Yaskawa INFORM job: sDrill44_(11).JBI

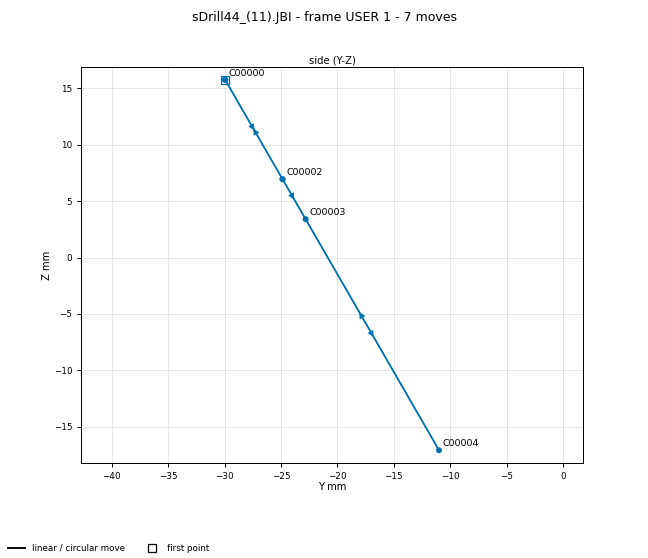
[picture p0: tool path of sDrill44_(11).JBI in frame USER 1, 7 of 7 moves have a stored position in this frame; points joined in program order, loops and branches not executed]
/JOB
//NAME sDrill44_(11)
//POS
///NPOS 7,0,0,0,0,0
///USER 1
///TOOL 3
///POSTYPE USER
///RECTAN
///RCONF 1,0,0,0,0,0
C00000=1.964,-29.946,15.742,-90.000,-150.794,-116.565
C00001=1.964,-29.946,15.742,-90.000,-150.794,-116.565
C00002=1.964,-24.866,6.943,-90.000,-150.794,-116.565
C00003=1.964,-22.817,3.394,-90.000,-150.794,-116.565
C00004=1.964,-11.000,-17.074,-90.000,-150.794,-116.565
C00005=1.964,-24.866,6.943,-90.000,-150.794,-116.565
C00006=1.964,-29.946,15.742,-90.000,-150.794,-116.565
//INST
///ATTR SC,RW,RJ
////FRAME USER 1
///GROUP1 RB1
///LVARS 2,0,0,0,0,0,0,0
NOP
SET LB000 1
SET LB001 25
MOVJ C00000 VJ=17
' Cutting Move Starts
MOVL C00001 V=17 PL=LB000 ACC=LB001 DEC=LB001
MOVL C00002 V=17 PL=LB000 ACC=LB001 DEC=LB001
MOVL C00003 V=17 PL=LB000 ACC=LB001 DEC=LB001
MOVL C00004 V=7 PL=LB000 ACC=LB001 DEC=LB001
MOVL C00005 V=17 PL=LB000 ACC=LB001 DEC=LB001
' Rapid Move Starts
MOVL C00006 V=17 PL=LB000 ACC=LB001 DEC=LB001
' By Autodesk Fusion CAM 2.0.20494
' Tool = 3
' Spindle = 5000 RPM
' Set Position Level
' Set Acceleration
' Program Start
' First Toolpath Point
END
